# EPICS substitutions: IOCs/12id/iocBoot/ioc12ida2/asynRecord.substitutions
file "$(ASYN)/db/asynRecord.db"
{
pattern
{P        R         PORT    ADDR    OMAX  IMAX}
{12ida2:     asyn_1   serial1    0     256  256}
{12ida2:     asyn_2   serial2    0     256  256}
{12ida2:     asyn_3   serial3    0     256  256}
{12ida2:     asyn_4   serial4    0     256  256}
{12ida2:     asyn_5   serial5    0     256  256}
{12ida2:     asyn_6   serial6    0     256  256}
{12ida2:     asyn_7   serial7    0     256  256}
{12ida2:     asyn_8   serial8    0     256  256}
{12ida2:     asyn_9   serial9    0     256  256}
{12ida2:     asyn_10   serial10    0     256  256}
{12ida2:     asyn_11   serial11    0     256  256}
{12ida2:     asyn_12   serial12    0     256  256}
{12ida2:     asyn_13   serial13    0     256  256}
{12ida2:     asyn_14   serial14    0     256  256}
{12ida2:     asyn_15   serial15    0     256  256}
{12ida2:     asyn_16   serial16    0     256  256}

#{12ida2:     gpib1    gpib1      1    2600 2600}
}
